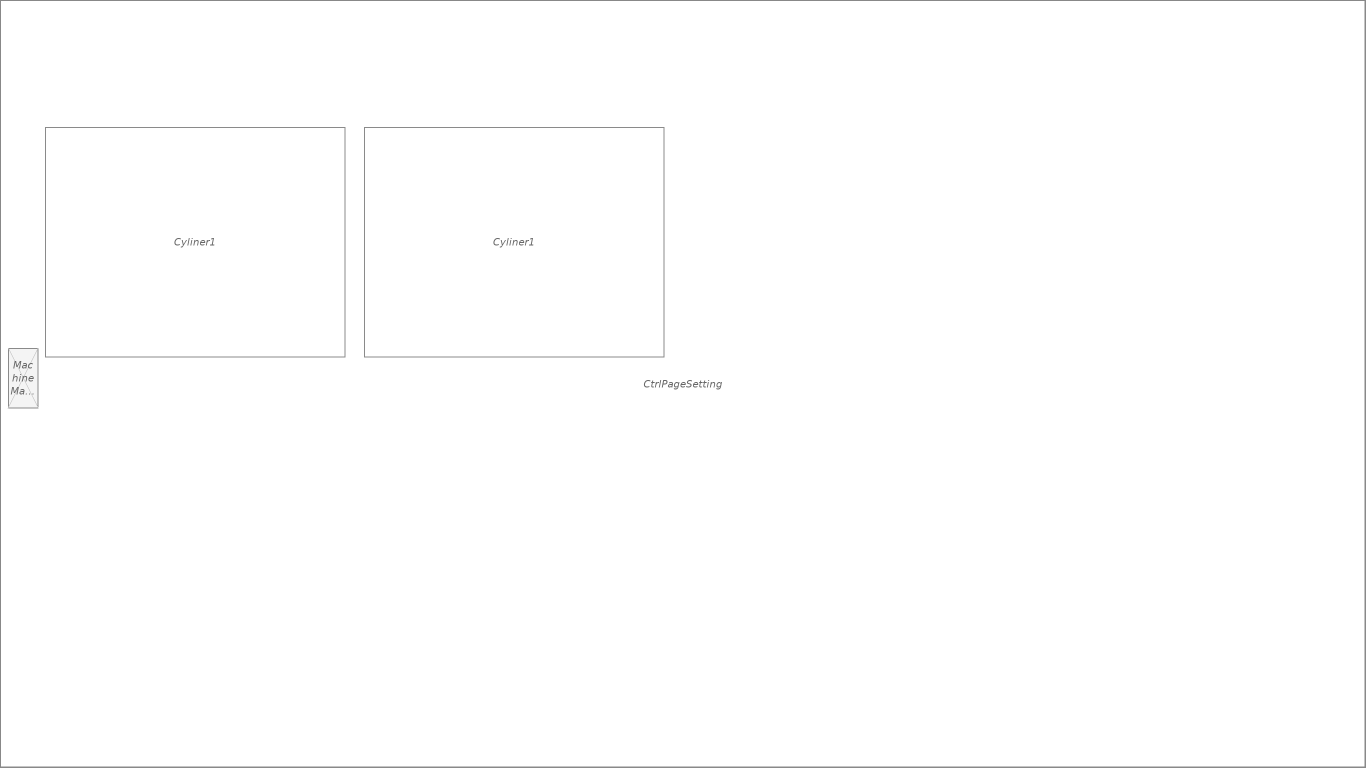
VISUALIZATION PageSetting_OpenLock_2  // 1366x768
    Frame (0,0 1366x768)
        shows CtrlPageSetting()
    Frame (45,127 300x230)
        shows Cyliner1(System := G_stSystem, Cylinder := G_arrCylinder[E_Cylinder.OpenLockPressPush], CylinderData := G_arrCylinderData[E_Cylinder.OpenLockPressPush])
    Frame (364,127 300x230)
        shows Cyliner1(System := G_stSystem, Cylinder := G_arrCylinder[E_Cylinder.OpenLockPressRotate], CylinderData := G_arrCylinderData[E_Cylinder.OpenLockPressRotate])
    Image (8,348 30x60), image: MachineManage.ImagePool.prev
        OnMouseClick: change screen: PageSetting_OpenLock
END_VISUALIZATION

(* stored: Version 1.1.0.1, ProductVersion 3.1.4024.3
   Visu PageSetting_OpenLock_2: Id {cdd4fce6-6dd4-43b6-aa8d-0360769a03eb} *)
